Staubli VAL3: TYPEDIO.pgx

public program typeDio(num pX, num pY, bool pTest)
begin
  //---------------------------------
  //  S H O W   S T A T U S   D I O
  //---------------------------------
  // Display the status of pTest
  //
  //  = true   "[x]"
  //  = false "[ ]"
  // See type()
  //---------------------------------
  // Staubli copyright 2003
  //                By CDIA 13 11 18
  //[Public]-------------------------
  //
  if (pTest==true)
    call type(pX,pY,"[x]")
  else
    call type(pX,pY,"[ ]")
  endIf
end
